INTERFACE ITF_BinarySensor

PROPERTY Value : BOOL
GET
END_GET
END_PROPERTY

END_INTERFACE

(* stored: Version 1.1.0.1
   Itf ITF_BinarySensor: Id {d7a604c8-0935-47a1-a540-ddbb35a9cad5}
   Property Value: Id {7f0ee423-7db7-467d-a10f-d968b6ef79b6}
   Get Get: Id {2172bd5f-5f30-4d38-b0ea-71b1681b96c4} *)
